TYPE ST_Actuatorstatus :
STRUCT
	AdvancedFeedback 	: BOOL;
	RetractedFeedback	: BOOL;
	Advancing			: BOOL;
	Retracting			: BOOL;
END_STRUCT
END_TYPE

(* stored: Version 1.1.0.1, ProductVersion 3.1.4024.12
   DUT ST_Actuatorstatus: Id {9106d7db-5025-4c30-805b-66c82597ebbd} *)
